(* LS Electric XG5000 project: Conveyer_Light_Control_System *)
(* PLC LSPLC *)
(* module base 0 slot 0: FEnet:XGL-EFMT(B) (Fast Ethernet 통신 모듈, 전기 Master) *)
(* module base 0 slot 1: 입력 모듈:XGI-D21A (DC 24V 입력, 8점 (전류소스/싱크입력)) *)
(* module base 0 slot 2: 출력 모듈:XGQ-RY1A (릴레이 출력, 8점 (2A용, 단독 COM.)) *)

(* Comments on direct variables
%MX0	기억용
%MX1	상승엣지 스캔
%MX2	램프 플리커 후 작동
%MX11	온오프 변화
*)

PROGRAM NewProgram (* task: 스캔 프로그램 *)
VAR
    C0 : CTD_INT;
    coil AT %IX0.0.3 : BOOL;
    Emergency_Stop AT %IX0.0.5 : BOOL;
    INT0 : INT := 0;
    OP_conveyer AT %QX0.1.0 : BOOL;
    OP_lamp AT %QX0.1.1 : BOOL;
    OP_Switch AT %IX0.0.0 : BOOL;
    reset : BOOL;
    search_defect AT %IX0.0.2 : BOOL;
    stop AT %IX0.0.1 : BOOL;
    T0 : TON;
    T1 : TON;
END_VAR

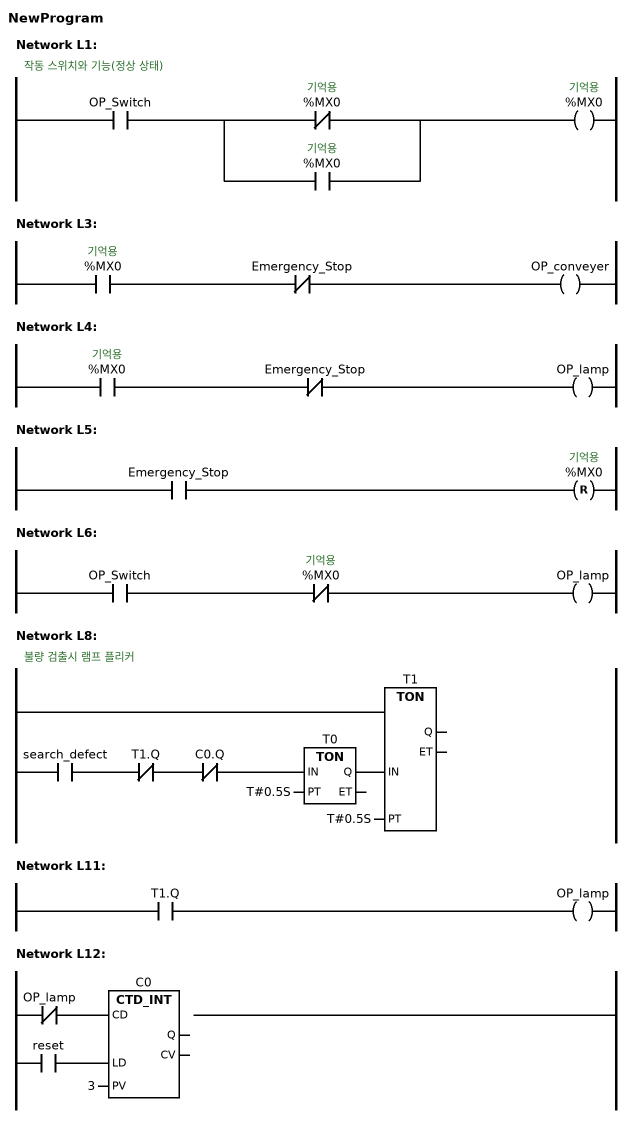
(* 작동 스위치와 기능(정상 상태) *)
(* Rung L1 *)
%MX0 := OP_Switch AND (NOT %MX0 OR %MX0);
(* Rung L3 *)
OP_conveyer := %MX0 AND NOT Emergency_Stop;
(* Rung L4 *)
OP_lamp := %MX0 AND NOT Emergency_Stop;
(* Rung L5 *)
IF Emergency_Stop THEN %MX0 := FALSE; END_IF;
(* Rung L6 *)
OP_lamp := OP_Switch AND NOT %MX0;
(* 불량 검출시 램프 플리커 *)
(* Rung L8 *)
T0(IN := search_defect AND NOT T1.Q AND NOT C0.Q, PT := T#0.5S);
T1(IN := T0.Q, PT := T#0.5S);
(* Rung L11 *)
OP_lamp := T1.Q;
(* Rung L12 *)
C0(CD := NOT OP_lamp, LD := reset, PV := 3);
END_PROGRAM

PROGRAM NEW (* task: 스캔 프로그램 *)
VAR
    C0 : CTU_INT;
    CV : INT;
    Emergency_Stop AT %IX0.0.1 : BOOL;
    OP_conveyer AT %QX0.1.0 : BOOL;
    OP_lamp AT %QX0.1.1 : BOOL;
    OP_lamp2 AT %QX0.1.2 : BOOL;
    OP_Switch AT %IX0.0.0 : BOOL;
    reset AT %IX0.0.3 : BOOL;
    search_defect AT %IX0.0.2 : BOOL;
    T0 : TON;
    T1 : TON;
END_VAR
VAR
    _e1 : R_TRIG;
END_VAR

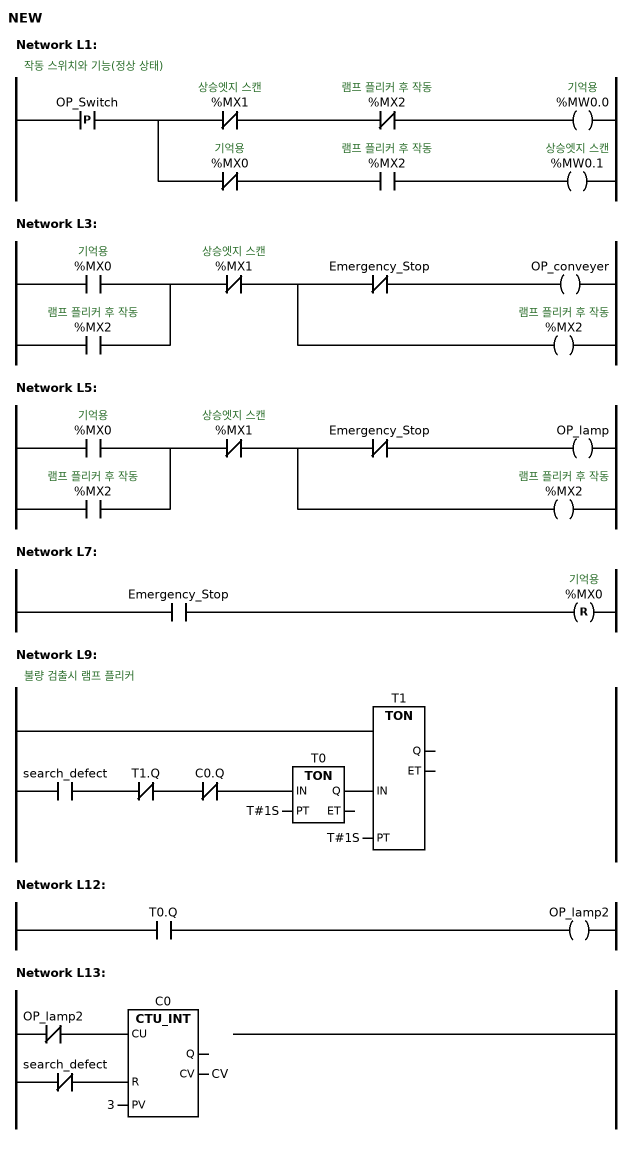
(* 작동 스위치와 기능(정상 상태) *)
(* Rung L1 *)
_e1(CLK := OP_Switch);
%MW0.0 := _e1.Q AND NOT %MX1 AND NOT %MX2;
%MW0.1 := _e1.Q AND NOT %MX0 AND %MX2;
(* Rung L3 *)
OP_conveyer := (%MX0 OR %MX2) AND NOT %MX1 AND NOT Emergency_Stop;
%MX2 := (%MX0 OR %MX2) AND NOT %MX1;
(* Rung L5 *)
OP_lamp := (%MX0 OR %MX2) AND NOT %MX1 AND NOT Emergency_Stop;
%MX2 := (%MX0 OR %MX2) AND NOT %MX1;
(* Rung L7 *)
IF Emergency_Stop THEN %MX0 := FALSE; END_IF;
(* 불량 검출시 램프 플리커 *)
(* Rung L9 *)
T0(IN := search_defect AND NOT T1.Q AND NOT C0.Q, PT := T#1S);
T1(IN := T0.Q, PT := T#1S);
(* Rung L12 *)
OP_lamp2 := T0.Q;
(* Rung L13 *)
C0(CU := NOT OP_lamp2, R := NOT search_defect, PV := 3, CV => CV);
END_PROGRAM